(* Logix 5000 project; controller CeramicPress Emulate 5570 rev 30.12; software revision 30.00 *)

TASK MainTask (continuous, watchdog 500 ms) : MainProgram

MODULES
   Local : Emulate 5570 (ICP 2, rev 30.12)
END_MODULES

PROGRAM MainProgram   (* main routine MainRoutine *)
VAR
   Action_000 : SFC_ACTION := (Status := 16#0020_0000, PauseTimer := 1);
   Action_001 : SFC_ACTION := (Status := 16#0020_0000, PauseTimer := 1);
   Action_002 : SFC_ACTION := (Status := 16#0020_0000, PauseTimer := 1);
   Action_003 : SFC_ACTION := (Status := 16#0020_0000, PauseTimer := 1);
   Action_004 : SFC_ACTION := (Status := 16#0020_0000, PauseTimer := 1);
   Action_005 : SFC_ACTION := (Status := 16#0020_0000, PauseTimer := 1);
   Action_006 : SFC_ACTION := (Status := 16#0020_0000, PauseTimer := 1);
   Action_007 : SFC_ACTION := (Status := 16#0020_0000, PauseTimer := 1);
   ActLX : REAL;
   ActLY : REAL;
   Manguera : BOOL;
   Step_000 : SFC_STEP := (Status := 16#0020_0000, PauseTimer := 1);
   Step_001 : SFC_STEP := (Status := 16#0020_0000, PauseTimer := 1);   // Mover hopper en x+
   Step_002 : SFC_STEP := (Status := 16#0020_0000, PauseTimer := 1);
   Step_003 : SFC_STEP := (Status := 16#0020_0000, PauseTimer := 1);   // Mover hopper en x-
   Step_004 : SFC_STEP := (Status := 16#0020_0000, PauseTimer := 1);
   Step_005 : SFC_STEP := (Status := 16#0020_0000, PauseTimer := 1);
   Step_006 : SFC_STEP := (Status := 16#0020_0000, PauseTimer := 1);
   Step_007 : SFC_STEP := (Status := 16#0020_0000, PauseTimer := 1);
   Step_008 : SFC_STEP := (Status := 16#0020_0000, PauseTimer := 1);
   Step_009 : SFC_STEP := (Status := 16#0020_0000, PauseTimer := 1);
   Step_010 : SFC_STEP := (Status := 16#0020_0000, PauseTimer := 1);
   Step_011 : SFC_STEP := (Status := 16#0020_0000, PauseTimer := 1);
   Tran_000 : BOOL;
   Tran_001 : BOOL;
   Tran_002 : BOOL;
   Tran_003 : BOOL;
   Tran_004 : BOOL;
   Tran_005 : BOOL;
   Tran_006 : BOOL;
   Tran_007 : BOOL;
   Tran_008 : BOOL;
   Xmax : BOOL;
   Xmin : BOOL;
END_VAR

ROUTINE Ceramic_Press   (* sequential function chart *)
// Ceramic Press Logic
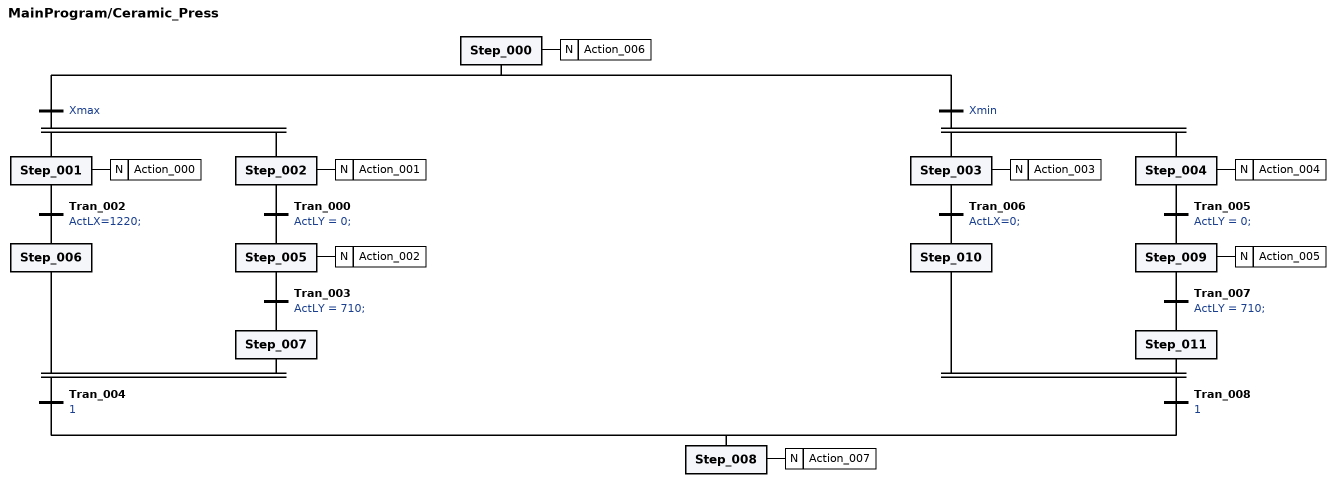
   STEP Step_000:
      ACTION Action_006 (N):
         Manguera :=1;
      END_ACTION
   END_STEP
   TRANSITION Xmax FROM Step_000 TO (Step_002, Step_001)
      := Xmax
   END_TRANSITION
   TRANSITION Xmin FROM Step_000 TO (Step_004, Step_003)
      := Xmin
   END_TRANSITION
   STEP Step_001:
      ACTION Action_000 (N):
         ActLX := 1220;
      END_ACTION
   END_STEP
   STEP Step_002:
      ACTION Action_001 (N):
         ActLY := 0;
      END_ACTION
   END_STEP
   STEP Step_003:
      ACTION Action_003 (N):
         ActLX := 0;
      END_ACTION
   END_STEP
   STEP Step_004:
      ACTION Action_004 (N):
         ActLY := 0;
      END_ACTION
   END_STEP
   TRANSITION Tran_002 FROM Step_001 TO Step_006
      := ActLX=1220;
   END_TRANSITION
   TRANSITION Tran_000 FROM Step_002 TO Step_005
      := ActLY = 0;
   END_TRANSITION
   TRANSITION Tran_006 FROM Step_003 TO Step_010
      := ActLX=0;
   END_TRANSITION
   TRANSITION Tran_005 FROM Step_004 TO Step_009
      := ActLY = 0;
   END_TRANSITION
   STEP Step_005:
      ACTION Action_002 (N):
         ActLY := 710;
         
      END_ACTION
   END_STEP
   STEP Step_009:
      ACTION Action_005 (N):
         ActLY := 710;
         
      END_ACTION
   END_STEP
   TRANSITION Tran_003 FROM Step_005 TO Step_007
      := ActLY = 710;
   END_TRANSITION
   TRANSITION Tran_007 FROM Step_009 TO Step_011
      := ActLY = 710;
   END_TRANSITION
   STEP Step_006:
   END_STEP
   STEP Step_007:
   END_STEP
   STEP Step_010:
   END_STEP
   STEP Step_011:
   END_STEP
   TRANSITION Tran_008 FROM (Step_010, Step_011) TO Step_008
      := 1
   END_TRANSITION
   TRANSITION Tran_004 FROM (Step_006, Step_007) TO Step_008
      := 1
   END_TRANSITION
   STEP Step_008:
      ACTION Action_007 (N):
         Manguera :=0;
      END_ACTION
   END_STEP
END_ROUTINE

ROUTINE MainRoutine   (* ladder *)
END_ROUTINE
END_PROGRAM
